// Mitsubishi GX Works2 project: a3   PLC: Q02/Q02H

PROGRAM MAIN
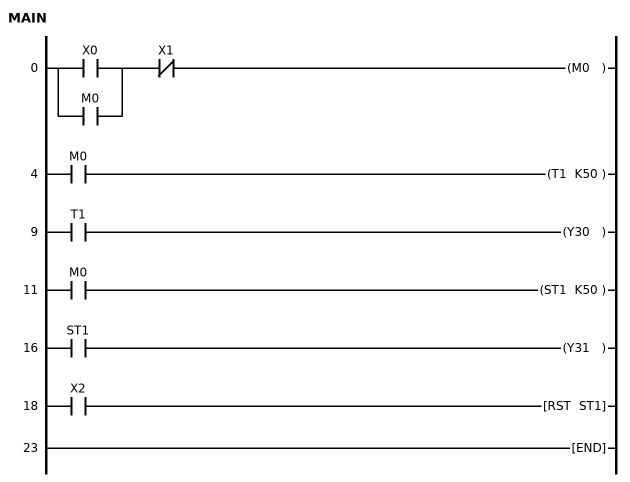
0     LD      X0
      OR      M0
      ANI     X1
      OUT     M0
4     LD      M0
      OUT     T1 K50
9     LD      T1
      OUT     Y30
11    LD      M0
      OUT     ST1 K50
16    LD      ST1
      OUT     Y31
18    LD      X2
      RST     ST1
23    END
END_PROGRAM
